(* IEC 61131-3 sources: programs/VI-54/VI-54_20171205/VI-54_20171205/Stations/Screen/LseClass170718/Class/StringBaseGB, 1 file *)

(* ---- StringBaseGB.st ---- *)
(*!
<Class
	Name               = "StringBaseGB"
	Revision           = "0.0"
	RealtimeTask       = "false"
	CyclicTask         = "false"
	BackgroundTask     = "true"
	Sigmatek           = "false"
	OSInterface        = "false"
	HighPriority       = "false"
	Automatic          = "false"
	UpdateMode         = "Prescan"
	SharedCommandTable = "true"
	Objectsize         = "(540,120)">
	<Channels>
	</Channels>
	<Network Name="StringBaseGB">
		<!-- List of Components in this network -->
		<Components>
			<Object
				Name       = "_base"
				Class      = "StringBase"
				Position   = "(218,120)"
				Visualized = "true">
				<Channels>
					<Server Name="Command"/>
					<Client Name="ToOsKernal"/>
				</Channels>
			</Object>
		</Components>
		<Comments>
		</Comments>
		<!-- List of Connections in this network -->
		<Connections>
			<Connection Source="this.Command" Destination="_base.Command" Vertices="(946,210),(774,210),"/>
		</Connections>
		<!-- Headerfiles -->
		<Options>
		</Options>
	</Network>
</Class>
*)
#pragma using StringBase

StringBaseGB : CLASS
: StringBase
  //Servers:
  //Clients:
  //Variables:
  //Functions:

	FUNCTION GLOBAL CalculateDigits
		VAR_INPUT
			Value 	: DINT;
		END_VAR
		VAR_OUTPUT
			Size 	: DINT;
		END_VAR;

	FUNCTION GLOBAL BuildValue2AsciiGB
		VAR_INPUT
			Value 	: DINT;
			pBaDest 	: ^CHAR;
			Offset 	: DINT;
		END_VAR
		VAR_OUTPUT
			Size 	: DINT;
		END_VAR;
  //Tables:
	FUNCTION @STD
		VAR_OUTPUT
			ret_code	: CONFSTATES;
		END_VAR;
	FUNCTION GLOBAL TAB @CT_;
END_CLASS;

FUNCTION GLOBAL StringBaseGB::CalculateDigits
	VAR_INPUT
		Value 	: DINT;
	END_VAR
	VAR_OUTPUT
		Size 	: DINT;
	END_VAR
  VAR
    ValueAbs : DINT;
  END_VAR

  Size := 1;

  if Value < 0 then
    Size += 1;
  end_if;

  ValueAbs := abs(Value);

  while ValueAbs > 9 do
    Size += 1;

    ValueAbs := ValueAbs / 10;
  end_while;

END_FUNCTION

FUNCTION GLOBAL StringBaseGB::BuildValue2AsciiGB
	VAR_INPUT
		Value 	: DINT;
		pBaDest 	: ^CHAR;
		Offset 	: DINT;
	END_VAR
	VAR_OUTPUT
		Size 	: DINT;
	END_VAR

  Size := BuildValue2Ascii(Value, CalculateDigits(Value), pBaDest, Offset);

END_FUNCTION
